// TIA Portal V18 export
FUNCTION_BLOCK "Seqencer"   // FB4, GRAPH
AUTHOR : dda
VERSION : 0.1
// stored: AcknowledgeErrorsRequired true, AutoNumber true, GraphVersion 6.0, InitialValuesAcquisition false, IsIECCheckEnabled true, LanguageInNetworks FBD, LockOperatingMode false, PermanentILProcessingInMANMode false, SetENOAutomatically true, SkipSteps false, UDAEnableTagReadback false, WithAlarmHandling true
   // inherited from GRAPH_BASE
   VAR
      OFF_SQ_BASE : Bool;
   END_VAR
   VAR_INPUT
      OFF_SQ { ExternalWritable := 'False'} : Bool := false;   // Turn sequence off
      INIT_SQ { ExternalWritable := 'False'} : Bool := false;   // Set sequence to initial state
      ACK_EF { ExternalWritable := 'False'} : Bool := false;   // Acknowledge all errors and faults
      REG_EF { ExternalWritable := 'False'} : Bool := false;   // Register all errors and faults
      ACK_S { ExternalWritable := 'False'} : Bool := false;   // Acknowledge step indicated in S_NO
      REG_S { ExternalWritable := 'False'} : Bool := false;   // Register the step indicated in S_NO
      HALT_SQ { ExternalWritable := 'False'} : Bool := false;   // Halt sequence immediately
      HALT_TM { ExternalWritable := 'False'} : Bool := false;   // Halt timers immediately
      ZERO_OP { ExternalWritable := 'False'} : Bool := false;   // Set all operands assigned with N, L, D to 0
      EN_IL { ExternalWritable := 'False'} : Bool := false;   // Enable interlocks
      EN_SV { ExternalWritable := 'False'} : Bool := false;   // Activate supervision processing
      EN_ACKREQ { ExternalWritable := 'False'} : Bool := false;   // Activate mandatory acknowledgment
      EN_SSKIP { ExternalWritable := 'False'} : Bool := false;   // Enable "Skip step"
      DISP_SACT { ExternalWritable := 'False'} : Bool := false;   // Display active steps only
      DISP_SEF { ExternalWritable := 'False'} : Bool := false;   // Display only steps with errors and disrupted steps
      DISP_SALL { ExternalWritable := 'False'} : Bool := false;   // Display all steps
      S_PREV { ExternalWritable := 'False'} : Bool := false;   // Output previous step in parameter S_NO
      S_NEXT { ExternalWritable := 'False'} : Bool := false;   // Indicate next step in parameter S_NO
      SW_AUTO { ExternalWritable := 'False'} : Bool := false;   // Automatic mode
      SW_TAP { ExternalWritable := 'False'} : Bool := false;   // Semiautomatic/switch with transition
      SW_TOP { ExternalWritable := 'False'} : Bool := false;   // Semiautomatic/ignore transition
      SW_MAN { ExternalWritable := 'False'} : Bool := false;   // Manual mode
      S_SEL { ExternalWritable := 'False'} : Int := 0;   // Select step to be output to S_NO
      S_SELOK { ExternalWritable := 'False'} : Bool := false;   // Enter value from S_SEL in S_NO
      S_ON { ExternalWritable := 'False'} : Bool := false;   // Activate step indicated in S_NO
      S_OFF { ExternalWritable := 'False'} : Bool := false;   // Disable step indicated in S_NO
      T_PREV { ExternalWritable := 'False'} : Bool := false;   // Display previous transition in T_NO
      T_NEXT { ExternalWritable := 'False'} : Bool := false;   // Display next transition at parameter T_NO
      T_PUSH { ExternalWritable := 'False'} : Bool := false;   // Enable transition to switch in semi automatic mode
      EN_LMODE { ExternalWritable := 'False'} : Bool := false;   // Activate learning mode
      RESET_CRIT { ExternalWritable := 'False'} : Bool := false;   // Reset all initial values recorded for interlocks and transitions
      startButton : Bool;
      lightBeam1 : Bool;
      lightBeam2 : Bool;
      lightBeam3 : Bool;
      robotArmDown : Bool;
      robotOnStation : Bool;
      robotOnMagazine : Bool;
      mySupervision : Bool;
   END_VAR
   VAR_OUTPUT
      S_NO { ExternalWritable := 'False'} : Int := 0;   // Step number
      S_MORE { ExternalWritable := 'False'} : Bool := false;   // More steps are available and can be shown in S_NO
      S_ACTIVE { ExternalWritable := 'False'} : Bool := false;   // Step indicated in S_NO is active
      S_TIME { ExternalWritable := 'False'} : Time := T#0ms;   // Step activation time
      S_TIMEOK { ExternalWritable := 'False'} : Time := T#0ms;   // No error in step activation time
      S_CRITLOC { ExternalWritable := 'False'} : DWord := 16#0;   // Interlock criteria bits
      S_CRITLOCERR { ExternalWritable := 'False'} : DWord := 16#0;   // Interlock criteria bits for event L1
      S_STATE { ExternalWritable := 'False'} : Word := 16#0;   // Step state bits
      T_NO { ExternalWritable := 'False'} : Int := 0;   // Transition number
      T_MORE { ExternalWritable := 'False'} : Bool := false;   // More valid transitions available for display
      T_CRIT { ExternalWritable := 'False'} : DWord := 16#0;   // Transition criteria bits
      T_CRITOLD { ExternalWritable := 'False'} : DWord := 16#0;   // Transition criteria bits from last cycle
      T_CRITFLT { ExternalWritable := 'False'} : DWord := 16#0;   // Transition criteria bits for event V1
      ERROR { ExternalWritable := 'False'} : Bool := false;   // Interlock group error
      FAULT { ExternalWritable := 'False'} : Bool := false;   // Supervision group error
      ERR_FLT { ExternalWritable := 'False'} : Bool := false;   // Interlock or supervision group error
      SQ_ISOFF { ExternalWritable := 'False'} : Bool := false;   // Sequence is off (no step active)
      SQ_HALTED { ExternalWritable := 'False'} : Bool := false;   // Sequence halted
      TM_HALTED { ExternalWritable := 'False'} : Bool := false;   // Timers halted
      OP_ZEROED { ExternalWritable := 'False'} : Bool := false;   // All the operands assigned with N, L, D are set to 0
      IL_ENABLED { ExternalWritable := 'False'} : Bool := false;   // Interlocks are active
      SV_ENABLED { ExternalWritable := 'False'} : Bool := false;   // Supervision processing activated
      ACKREQ_ENABLED { ExternalWritable := 'False'} : Bool := false;   // Mandatory acknowledgment activated
      SSKIP_ENABLED { ExternalWritable := 'False'} : Bool := false;   // Skip steps activated
      SACT_DISP { ExternalWritable := 'False'} : Bool := false;   // Display active steps only
      SEF_DISP { ExternalWritable := 'False'} : Bool := false;   // Display only steps with errors or disrupted steps
      SALL_DISP { ExternalWritable := 'False'} : Bool := false;   // Display all steps
      AUTO_ON { ExternalWritable := 'False'} : Bool := false;   // Automatic mode is active
      TAP_ON { ExternalWritable := 'False'} : Bool := false;   // Semiautomatic mode/step with transition enabled
      TOP_ON { ExternalWritable := 'False'} : Bool := false;   // Semiautomatic mode/ignore transition enabled
      MAN_ON { ExternalWritable := 'False'} : Bool := false;   // Manual mode is active
      LMODE_ENABLED { ExternalWritable := 'False'} : Bool := false;   // Learning mode is active
      partInPos1 { ExternalAccessible := 'False'; ExternalVisible := 'False'; ExternalWritable := 'False'} : Bool;
      partInPos2 { ExternalAccessible := 'False'; ExternalVisible := 'False'; ExternalWritable := 'False'} : Bool;
      partInPos3 { ExternalAccessible := 'False'; ExternalVisible := 'False'; ExternalWritable := 'False'} : Bool;
      startConv { ExternalAccessible := 'False'; ExternalVisible := 'False'; ExternalWritable := 'False'} : Bool;
      automaticMode { ExternalAccessible := 'False'; ExternalVisible := 'False'; ExternalWritable := 'False'} : Bool;
      robotFill { ExternalAccessible := 'False'; ExternalVisible := 'False'; ExternalWritable := 'False'} : Bool;
      robotGoToMagazine { ExternalAccessible := 'False'; ExternalVisible := 'False'; ExternalWritable := 'False'} : Bool;
      robotGoToStation { ExternalAccessible := 'False'; ExternalVisible := 'False'; ExternalWritable := 'False'} : Bool;
   END_VAR
   VAR
      statLightbeam3Fal { ExternalAccessible := 'False'; ExternalVisible := 'False'; ExternalWritable := 'False'} : Bool;
      statMemoryTag { ExternalAccessible := 'False'; ExternalVisible := 'False'; ExternalWritable := 'False'} : Bool;
   END_VAR
BEGIN
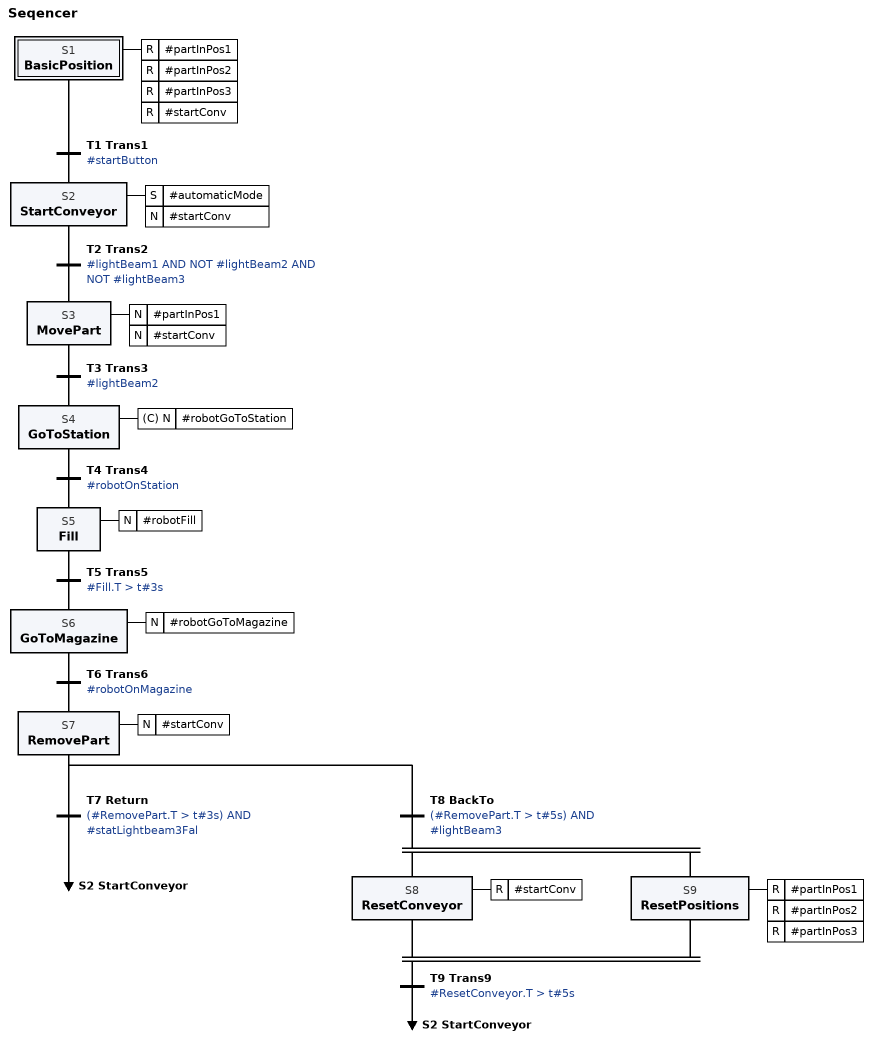
   // sequencer 1
   INITIAL_STEP BasicPosition:   // S1, max time T#10S, warning time T#7S
      supervision V := (#StartConveyor.T > t#10ms) AND (#StartConveyor.U > t#10ms);
              R    #partInPos1
              R    #partInPos2
              R    #partInPos3
              R    #startConv
   END_STEP
   TRANSITION Trans1 FROM BasicPosition TO StartConveyor   // T1
      := #startButton;
   END_TRANSITION
   STEP StartConveyor:   // S2, max time T#10S, warning time T#7S
              S    #automaticMode
              N    #startConv
   END_STEP
   TRANSITION Trans2 FROM StartConveyor TO MovePart   // T2
      := #lightBeam1 AND NOT #lightBeam2 AND NOT #lightBeam3;
   END_TRANSITION
   STEP MovePart:   // S3, max time T#10S, warning time T#7S
              N    #partInPos1
              N    #startConv
   END_STEP
   TRANSITION Trans3 FROM MovePart TO GoToStation   // T3
      := #lightBeam2;
   END_TRANSITION
   STEP GoToStation:   // S4, max time T#10S, warning time T#7S
      interlock C := NOT #robotArmDown;
      (C)     N    #robotGoToStation
   END_STEP
   TRANSITION Trans4 FROM GoToStation TO Fill   // T4
      := #robotOnStation;
   END_TRANSITION
   STEP Fill:   // S5, max time T#10S, warning time T#7S
              N    #robotFill
   END_STEP
   TRANSITION Trans5 FROM Fill TO GoToMagazine   // T5
      := #Fill.T > t#3s;
   END_TRANSITION
   STEP GoToMagazine:   // S6, max time T#10S, warning time T#7S
              N    #robotGoToMagazine
   END_STEP
   TRANSITION Trans6 FROM GoToMagazine TO RemovePart   // T6
      := #robotOnMagazine;
   END_TRANSITION
   STEP RemovePart:   // S7, max time T#10S, warning time T#7S
      supervision V := (#RemovePart.T < #RemovePart.T_MAX) AND (#RemovePart.T > #RemovePart.T_WARN);
              N    #startConv
   END_STEP
   TRANSITION "Return" FROM RemovePart TO StartConveyor   // T7, jump
      := (#RemovePart.T > t#3s) AND #statLightbeam3Fal;
   END_TRANSITION
   TRANSITION BackTo FROM RemovePart TO (ResetConveyor, ResetPositions)   // T8
      := (#RemovePart.T > t#5s) AND #lightBeam3;
   END_TRANSITION
   STEP ResetConveyor:   // S8, max time T#10S, warning time T#7S
              R    #startConv
   END_STEP
   STEP ResetPositions:   // S9, max time T#10S, warning time T#7S
      interlock C := #ResetPositions.T > #ResetPositions.T_MAX;
              R    #partInPos1
              R    #partInPos2
              R    #partInPos3
   END_STEP
   TRANSITION Trans9 FROM (ResetConveyor, ResetPositions) TO StartConveyor   // T9, jump
      := #ResetConveyor.T > t#5s;
   END_TRANSITION
END_FUNCTION_BLOCK
